// TIA Portal V17 export
// export: Created 2021-12-03T08:13:13.9954486Z, ExportSetting WithDefaults, DisplayName Totally Integrated Automation Portal, DisplayVersion V17, DisplayName TIA Portal Openness, DisplayVersion V17, DisplayName TIA Portal Version Control Interface, DisplayVersion V17, DisplayName STEP 7 Professional, DisplayVersion V17, DisplayName STEP 7 Safety, DisplayVersion V17, DisplayName WinCC Advanced, DisplayVersion V17
DATA_BLOCK "FDBI_Simulation"   // DB81, F_DB
VERSION : 0.1
// stored: AutoNumber false, InstanceOfName FFB_Simulation, InstanceOfType FB
"FFB_Simulation"
   // VAR
   //    SimEmSt { ExternalVisible := 'False'; ExternalWritable := 'False'} : Bool;
   //    SimEnd { ExternalVisible := 'False'; ExternalWritable := 'False'} : Bool;
   //    Empty : Bool;
   // END_VAR
BEGIN
END_DATA_BLOCK
